Omron CX-Programmer project NewProject (CX-Programmer 9.73)

# PLC NewPLC1: CP1E N20

## Global symbols (name address type ; comment)
0.01 BOOL  ; PB START
0.02 BOOL  ; PB STOP
100.01 BOOL  ; OUTPUT
100.02 BOOL  ; PB STOP

## Program NewProgram1 (cyclic task 0)

### Section Section1

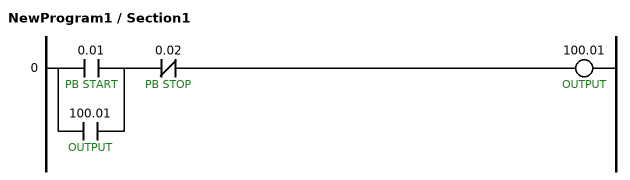
; rung 0
LD 0.01  ; PB START
OR 100.01  ; OUTPUT
ANDNOT 0.02  ; PB STOP
OUT 100.01  ; OUTPUT

### Section END
; rung 0
END(001)